FUNCTION_BLOCK FB_InfoMON
VAR_INPUT
	stInfoData 			:		DUT_ST_InfoDataFB ;
END_VAR
VAR_OUTPUT
	sState 				: 		STRING ;
	sDiag 				: 		STRING ;
	END_VAR
VAR
END_VAR

// Guard Door Monitor FB's State
IF stInfoData.usiMapState 			= 	0 THEN
				sState 				:= 	'Undefined' ;
	ELSIF stInfoData.usiMapState 	= 	1 THEN
				sState 				:= 	'RUN' ;
	ELSIF stInfoData.usiMapState 	= 	2 THEN
				sState 				:= 	'STOP' ;
	ELSIF stInfoData.usiMapState 	= 	3 THEN
				sState 				:= 	'SAFE' ;
	ELSIF stInfoData.usiMapState 	= 	4 THEN
				sState 				:= 	'ERROR' ;
	ELSIF stInfoData.usiMapState 	= 	5 THEN
				sState 				:= 	'RESET' ;
	ELSIF stInfoData.usiMapState 	= 	6 THEN
				sState				:= 	'START' ;
	ELSIF stInfoData.usiMapState 	= 	7 THEN
				sState 				:= 	'Error Delay' ;
	ELSIF stInfoData.usiMapState 	= 	8 THEN
				sState 				:= 	'DelayOut' ;
	ELSIF stInfoData.usiMapState 	= 	9 THEN
				sState 				:= 	'Function Test' ;
	ELSE
				sState 				:= 	'Unknown' ;
END_IF

// Guard Door Monitor FB's Diagnostics
IF stInfoData.uiMapDiag 			= 	0 THEN
				sDiag 				:= 	'No Error' ;
ELSIF  stInfoData.uiMapDiag 		= 	1 THEN
				sDiag 				:= 	'Discrepancy Error of Input Group 1' ;
ELSIF  stInfoData.uiMapDiag 		= 	2 THEN
				sDiag 				:= 	'Discrepancy Error of Input Group 2' ;
ELSIF  stInfoData.uiMapDiag 		= 	4 THEN
				sDiag 				:= 	'Discrepancy Error of the Secure Inputs' ;
ELSIF  stInfoData.uiMapDiag 		= 	16 THEN
				sDiag 				:= 	'EDM 1 Monitoring Error' ;
ELSIF  stInfoData.uiMapDiag 		= 	32 THEN
				sDiag 				:= 	'EDM 2 Monitoring Error' ;
ELSE
				sDiag 				:= 	'Unknown' ;
END_IF

END_FUNCTION_BLOCK

(* stored: Version 1.1.0.1, ProductVersion 3.1.0.14
   POU FB_InfoMON: Id {b90b6e11-248d-4ce7-be92-0402ccbcc515} *)
